(*

.. <legal notes>

legal notes
=================
| SPDX-FileCopyrightText: © 2026 Oleksandr Tiutyk <trofimich@gmail.com>
| SPDX-License-Identifier: LGPL-3.0-only
| For details check: LGPL-3.0-only_

.. _LGPL-3.0-only: https://www.gnu.org/licenses/lgpl-3.0.en.html

.. </legal notes>

*)

{attribute 'no_explicit_call' := 'do not call this function block directly'} 
{attribute 'enable_dynamic_creation'}
// Collection of bytes of dynamic size
FUNCTION_BLOCK DynamicByteList EXTENDS Core.Object IMPLEMENTS IDynamicByteList
VAR_OUTPUT
	DataAddress : POINTER TO BYTE;
END_VAR
VAR
	_ClassName : STRING := __POUNAME();
	
	_Capacity : DINT;
	_Length : DINT;
END_VAR

METHOD AppendAny : IDynamicByteList
VAR_INPUT
	data : ANY;
END_VAR
AppendAny := AppendData(data.pValue, TO_UDINT(data.diSize));
END_METHOD

METHOD AppendByte : IDynamicByteList
VAR_INPUT
	value : BYTE;
END_VAR
VAR
	newMemory : POINTER TO BYTE;
END_VAR
AppendByte := AppendData(ADR(value), 1);
END_METHOD

METHOD AppendData : IDynamicByteList
VAR_INPUT
	data : POINTER TO BYTE;
	dataSize : UDINT;
END_VAR
VAR
	newMemory : POINTER TO BYTE;
END_VAR
AppendData := THIS^;

IF data = 0 OR_ELSE dataSize = 0 THEN
	RETURN;
END_IF

// if existing memory is not enough
IF _Length + TO_DINT(dataSize) > _Capacity THEN
	// calculate new memory size
	_Capacity := _Length + TO_DINT(dataSize);
	
	// allocate new memory
	newMemory := __NEW(BYTE, TO_UDINT(_Capacity));
	
	// copy existing bytes to new memory if needed
	IF _Length > 0 THEN
		Tc2_System.MEMCPY(newMemory, DataAddress, TO_UDINT(_Length));		
	END_IF
	
	// release old memory
	IF DataAddress <> 0 THEN
		__DELETE(DataAddress);		
	END_IF
	
	// save new memory reference
	DataAddress := newMemory;
END_IF

// append new bytes
Tc2_System.MEMCPY(DataAddress + TO_DWORD(_Length), data, dataSize);

// set new bytes count
_Length := _Length + TO_DINT(dataSize);
END_METHOD

METHOD AppendGeneric : IDynamicByteList
VAR_INPUT
	data : Core.GENERIC_VALUE;
END_VAR
AppendGeneric := AppendData(data.Address, TO_UDINT(data.Size));
END_METHOD

{attribute 'monitoring' := 'call'}
PROPERTY FINAL Capacity : COLLECTION_LENGTH
GET
Capacity := _Capacity;
END_GET
END_PROPERTY

{attribute 'monitoring' := 'call'}
PROPERTY ClassName : STRING
GET
ClassName := _ClassName;
END_GET
END_PROPERTY

METHOD Clear : IDynamicByteList
VAR_INPUT
	releaseMemory : BOOL := FALSE;
END_VAR
Clear := THIS^;

IF releaseMemory AND_THEN _Capacity > 0 THEN
	__DELETE(DataAddress);
	_Capacity := 0;
END_IF

_Length := 0;
END_METHOD

METHOD CreateEnumerator : IEnumerator
VAR
	enumerator : POINTER TO DynamicByteListEnumerator;
END_VAR
enumerator := __NEW(DynamicByteListEnumerator(list := THIS^));

CreateEnumerator := enumerator^;
END_METHOD

{attribute 'monitoring' := 'call'}
PROPERTY FINAL Empty : BOOL
GET
Empty := _Length <= 0;
END_GET
END_PROPERTY

METHOD FB_exit : BOOL
VAR_INPUT
	bInCopyCode : BOOL; // if TRUE, the exit method is called for exiting an instance that is copied afterwards (online change).
END_VAR
Clear(TRUE);
END_METHOD

METHOD Find : BOOL
VAR_INPUT
	value : BYTE;
END_VAR
VAR_OUTPUT
	index : COLLECTION_INDEX;
END_VAR
VAR
	i : DINT;	
END_VAR
IF _Length > 0 THEN
	FOR i := 0 TO _Length - 1 DO
		IF DataAddress[i] = value THEN
			index := i;
			Find := TRUE;
			RETURN;
		END_IF 	
	END_FOR
END_IF
END_METHOD

METHOD Get : BYTE
VAR_INPUT
	index : COLLECTION_INDEX;
END_VAR
VAR
	exception : StandardException;
END_VAR
IF DataAddress = 0 THEN
	exception.ThrowByObject(THIS^, __POUNAME(), __POSITION(), "Dynamic byte array is empty");
END_IF

IF index < 0 THEN
	exception.ThrowByObject(THIS^, __POUNAME(), __POSITION(), "Index is less then zero");
END_IF

IF index >= _Length THEN
	exception.ThrowByObject(THIS^, __POUNAME(), __POSITION(), "Index is too large");
END_IF

Get := DataAddress[index];
END_METHOD

{attribute 'monitoring' := 'call'}
PROPERTY FINAL Length : COLLECTION_LENGTH
GET
Length := _Length;
END_GET
END_PROPERTY

METHOD LoadFromAny : IDynamicByteList
VAR_INPUT
	data : ANY;
	startIndex : COLLECTION_INDEX := 0;
END_VAR
LoadFromAny := LoadFromData(data.pValue, TO_ULINT(data.diSize), startIndex);
END_METHOD

METHOD LoadFromData : IDynamicByteList
VAR_INPUT
	data : POINTER TO BYTE;
	dataSize : ULINT;
	startIndex : COLLECTION_INDEX := 0;
END_VAR
VAR
	exception : Core.ArgumentOutOfRangeException;
	
	newMemory : POINTER TO BYTE;
END_VAR
IF TO_DINT(startIndex) > _Length THEN
	exception.ThrowByObject(THIS^, __POUNAME(), __POSITION(), 'startIndex', startIndex);
END_IF

IF dataSize < 0 THEN
	exception.ThrowByObject(THIS^, __POUNAME(), __POSITION(), 'dataSize', dataSize);
END_IF

LoadFromData := THIS^;
 
IF data = 0 OR_ELSE dataSize = 0 THEN
	RETURN;
END_IF

IF startIndex + TO_DINT(dataSize) > _Capacity THEN
	// calculate new memory size
	_Capacity := startIndex + TO_DINT(dataSize);
	
	// allocate new memory
	newMemory := __NEW(BYTE, TO_UDINT(_Capacity));
	
	// copy existing bytes to new memory if needed
	IF startIndex > 0 THEN
		Tc2_System.MEMCPY(newMemory, DataAddress, TO_UDINT(startIndex));		
	END_IF
	
	// append new bytes
	Tc2_System.MEMCPY(newMemory + TO_DWORD(startIndex), data, TO_UDINT(dataSize));
	
	// set new bytes count
	_Length := _Capacity;
	
	// release old memory
	IF DataAddress <> 0 THEN
		__DELETE(DataAddress);		
	END_IF
	
	// save new memory reference
	DataAddress := newMemory;
ELSE
	// append new bytes
	Tc2_System.MEMCPY(dataAddress + TO_DWORD(startIndex), data, TO_UDINT(dataSize));
	
	// set new bytes count
	_Length := startIndex + TO_DINT(dataSize);	
END_IF
END_METHOD

METHOD LoadFromGeneric : IDynamicByteList
VAR_INPUT
	data : Core.GENERIC_VALUE;
	startIndex : COLLECTION_INDEX := 0;
END_VAR
LoadFromGeneric := LoadFromData(data.Address, data.Size, startIndex);
END_METHOD

{attribute 'monitoring' := 'call'}
PROPERTY NamespaceName : STRING
GET
NamespaceName := CurrentNamespace.Name;
END_GET
END_PROPERTY

METHOD Remove : IDynamicByteList
VAR_INPUT
	value : BYTE;
END_VAR
VAR
	index : DINT;
	exception : StandardException;
END_VAR
IF DataAddress = 0 THEN
	exception.ThrowByObject(THIS^, __POUNAME(), __POSITION(), "Dynamic byte array is empty");
END_IF

IF Length < 0 THEN
	exception.ThrowByObject(THIS^, __POUNAME(), __POSITION(), "Count is less then zero");
END_IF

IF index + Length > _Length THEN
	exception.ThrowByObject(THIS^, __POUNAME(), __POSITION(), "Index + count are outside the array bounds");
END_IF

Remove := THIS^;

IF Find(value, index => index) THEN
	RemoveAt(index, 1);
END_IF
END_METHOD

METHOD RemoveAt : IDynamicByteList
VAR_INPUT
	index : COLLECTION_INDEX;
	count : COLLECTION_LENGTH := 1;
END_VAR
VAR
	exception : StandardException;
	newMemory : POINTER TO BYTE;
END_VAR
IF DataAddress = 0 THEN
	exception.ThrowByObject(THIS^, __POUNAME(), __POSITION(), "Dynamic byte array is empty");
END_IF

IF index < 0 THEN
	exception.ThrowByObject(THIS^, __POUNAME(), __POSITION(), "Index is less then zero");
END_IF

IF count < 0 THEN
	exception.ThrowByObject(THIS^, __POUNAME(), __POSITION(), "Count is less then zero");
END_IF

IF index + count > _Length THEN
	exception.ThrowByObject(THIS^, __POUNAME(), __POSITION(), "Index + count are outside the array bounds");
END_IF

RemoveAt := THIS^;

// calculate new memory size
_Capacity := _Length - count;

// allocate new memory
newMemory := __NEW(BYTE, TO_UDINT(_Capacity)); 

// copy leading bytes if needed
IF index <> 0 THEN
	Tc2_System.MEMCPY(newMemory, DataAddress, TO_UDINT(index));
END_IF

// copy trailing bytes
Tc2_System.MEMCPY(newMemory + TO_DWORD(index), DataAddress + TO_DWORD(index + count), TO_UDINT(_Length - index - count));

// release old buffer
__DELETE(DataAddress);

// save new buffer
DataAddress := newMemory;

// set bytes count
_Length := _Capacity;
END_METHOD

METHOD Resize : IDynamicByteList
VAR_INPUT
	newBytesCount : DINT; 
END_VAR
VAR
	exception : StandardException;
	newMemory : POINTER TO BYTE;
END_VAR
IF newBytesCount < 0 THEN
	exception.ThrowByObject(THIS^, __POUNAME(), __POSITION(), "New bytes count is less then zero");
END_IF

Resize := THIS^;

// if existing memory is not enough
IF newBytesCount > _Capacity THEN
	// calculate new memory size
	_Capacity := newBytesCount;
	
	// allocate new memory
	newMemory := __NEW(BYTE, TO_UDINT(_Capacity));
	
	// copy existing bytes to new memory if needed
	IF _Length > 0 THEN
		Tc2_System.MEMCPY(newMemory, DataAddress, TO_UDINT(_Length));		
	END_IF
	
	// release old memory
	IF DataAddress <> 0 THEN
		__DELETE(DataAddress);		
	END_IF
	
	// save new memory reference
	DataAddress := newMemory;
END_IF

// set new bytes count
_Length := newBytesCount;
END_METHOD

{attribute 'monitoring' := 'call'}
PROPERTY SelfSize : ULINT
GET
SelfSize := XSIZEOF(THIS^);
END_GET
END_PROPERTY

METHOD Set : IDynamicByteList
VAR_INPUT
	index : COLLECTION_INDEX;
	value : BYTE;
END_VAR
VAR
	exception : StandardException;
END_VAR
IF DataAddress = 0 THEN
	exception.ThrowByObject(THIS^, __POUNAME(), __POSITION(), "Dynamic byte array is empty");
END_IF

IF index < 0 THEN
	exception.ThrowByObject(THIS^, __POUNAME(), __POSITION(), "Index is less then zero");
END_IF

IF index >= _Length THEN
	exception.ThrowByObject(THIS^, __POUNAME(), __POSITION(), "Index is too large");
END_IF

Set := THIS^;

DataAddress[index] := value;
END_METHOD

END_FUNCTION_BLOCK

(* stored: Version 1.1.0.1
   POU DynamicByteList: Id {44085af7-7241-03f1-3e6d-aeb87f0c58dd}, SpecialFunc None
   Method AppendAny: Id {fa939ac2-b614-4bc3-8ef3-f524865ffb5f}
   Method AppendByte: Id {90a35576-aaee-0fbc-214a-d1c0f81c72fb}
   Method AppendData: Id {d35c3ee4-7daa-49d5-be43-e476b3efb046}
   Method AppendGeneric: Id {ac72fb80-d130-4ae7-81e5-86ab3708db48}
   Property Capacity: Id {39da2e53-b31d-4366-b174-c1e7fcd2d73a}
   Get Get: Id {e45b1a1e-b7c6-4e97-befa-5db022de37f9}
   Property ClassName: Id {3b9bf934-b83c-0948-370d-5e8e28db661a}
   Get Get: Id {a74d6b23-00f3-0fef-283c-b96c5cad2f8b}
   Method Clear: Id {58795b0c-c9a9-0b7d-1801-4867f25906b7}
   Method CreateEnumerator: Id {9eb1bbc5-e145-4b1d-be02-fc14e3a7b7c4}
   Property Empty: Id {8cac260d-f211-4946-9f91-204b369e9bc6}
   Get Get: Id {cdc3f172-a10e-45a6-be1f-94a4244848e7}
   Method FB_exit: Id {58cee31c-ede5-0b41-17b5-f6dfb8c1dea7}
   Method Find: Id {f870e801-4961-0438-0486-eeff60dc3fea}
   Method Get: Id {7a2d32dc-2bf1-07fe-3b69-aed2ad5b300d}
   Property Length: Id {d1b0052d-4e1b-09cb-235e-e87df6b9b5a5}
   Get Get: Id {457f3f94-ecd5-03a2-1012-5eb779d04c66}
   Method LoadFromAny: Id {6ca12394-c5fc-0274-1ee4-d0bfc0727c06}
   Method LoadFromData: Id {9fe65b5e-87b5-0537-23bd-6a15d825d74e}
   Method LoadFromGeneric: Id {803d0535-a6e1-4d89-878a-9e90b4d80911}
   Property NamespaceName: Id {6affa192-b708-4407-b07b-3f99b221293a}
   Get Get: Id {08e774db-64ad-4b08-8c9f-7cf3351a9ee4}
   Method Remove: Id {bf82b30e-92dd-0d23-0038-cce05024df18}
   Method RemoveAt: Id {13c7901e-f730-033f-2407-dd64a3fc2480}
   Method Resize: Id {8b327940-8027-042d-2b0a-ccea3f4d165c}
   Property SelfSize: Id {eb116396-1c6b-495f-b284-5b142fa86f6c}
   Get Get: Id {9d568fff-ebc6-4d27-9dd9-94ca65277b07}
   Method Set: Id {7b62d34d-7ee9-07a4-2e13-b032abd0cd09} *)
